(* PLC project  *)

PROGRAM P

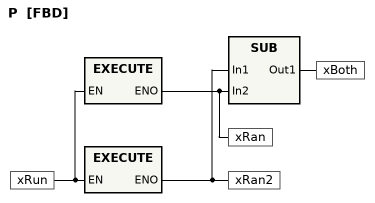
(* FBD diagram, written out as Structured Text *)
IF xRun THEN
  nCount := nCount + 1;
END_IF;
IF xRun THEN
  nOther := nOther + 2;
END_IF;
xRan := xRun;
xRan2 := xRun;
xBoth := xRun - xRun;
END_PROGRAM
